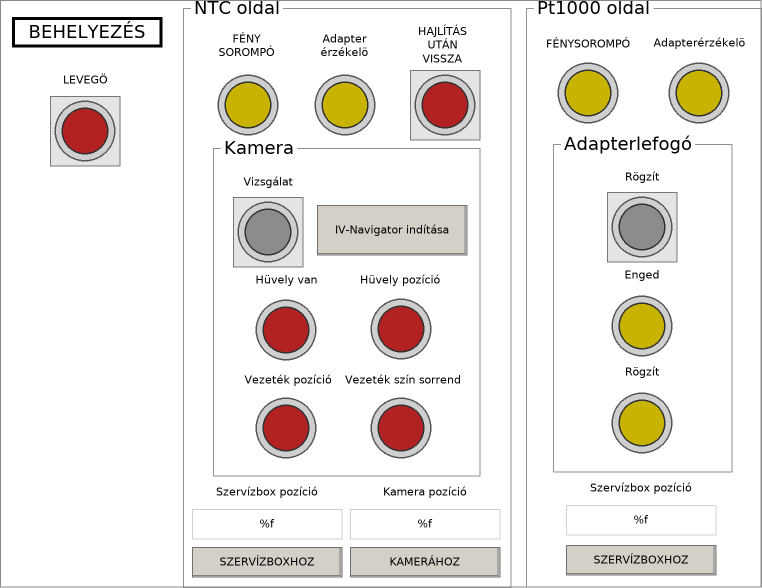
VISUALIZATION Behelyezes  // 762x588
    GroupBox (526,0 236x587), "Pt1000 oldal"
        GroupBox (27,136 179x336), "Adapterlefogó"
            PushSwitch (54,56 70x70), variable: GVL.bAdapterLefogo, behaviour: TOGGLE, style: Switch-PushSwitch-Gray
            Lamp1 (54,155 70x70), variable: GVL.bAdapterLefogoBent, style: Lamp-Lamp1-Yellow
            Lamp1 (54,252 70x70), variable: GVL.bAdapterLefogoKint, style: Lamp-Lamp1-Yellow
            Label (61,226 57x20), "Rögzít"
            Label (62,129 54x20), "Enged"
            Label (60,31 59x20), "Rögzít"
        Lamp1 (138,58 70x70), variable: GVL.bAdaptererzekelo, style: Lamp-Lamp1-Yellow
        Label (122,33 103x20), "Adapterérzékelö"
        Lamp1 (27,58 70x70), variable: GVL.bFenysorompoPt, style: Lamp-Lamp1-Yellow
        Label (10,34 104x20), "FÉNYSOROMPÓ"
        Group (40,478 150x97)
            Button (0,67 150x30), "SZERVÍZBOXHOZ"
                OnMouseUp: execute { PISTITENGELY.lrPistiPosition:=GVL.lrPtSzervizbox; PISTITENGELY.sPistiAxisCommand:='MOVE'; }
            Textfield (0,27 150x30), "%f", text variable: GVL.lrPtSzervizbox
                OnMouseClick: write the text variable via VisuDialogs.Numpad, min -10000, max -1
            Label (0,0 150x20), "Szervízbox pozíció"
    RoundedRectangle (12,17 150x30)
    Label (12,17 150x30), "BEHELYEZÉS"
    GroupBox (183,0 328x588), "NTC oldal"
        GroupBox (30,140 267x336), "Kamera"
            Group (20,32 70x95)
                PushSwitch (0,25 70x70), variable: GVL.bKameraTrigger, behaviour: TOGGLE, style: Switch-PushSwitch-Gray
                Label (2,0 67x20), "Vizsgálat"
            Lamp1 (153,154 70x70), variable: GVL.bKameraHulsePozOK, style: Lamp-Lamp1-Green
            Lamp1 (153,253 70x70), variable: GVL.bKameraSzinekOK, style: Lamp-Lamp1-Green
            Label (130,230 120x20), "Vezeték szín sorrend"
            Label (140,130 94x20), "Hüvely pozíció"
            Lamp1 (153,154 70x70), variable: NOT GVL.bKameraHulsePozOK, invisible if: NOT KAMERA.bVizsgalatKesz OR GVL.bKameraHulsePozOK, style: Lamp-Lamp1-Red
            Lamp1 (153,253 70x70), variable: NOT GVL.bKameraSzinekOK, invisible if: NOT KAMERA.bVizsgalatKesz OR GVL.bKameraSzinekOK, style: Lamp-Lamp1-Red
            Label (30,230 90x20), "Vezeték pozíció"
            Lamp1 (38,253 70x70), variable: GVL.bKameraVezetekPozOK, style: Lamp-Lamp1-Green
            Lamp1 (38,253 70x70), variable: NOT GVL.bKameraVezetekPozOK, invisible if: NOT KAMERA.bVizsgalatKesz OR GVL.bKameraVezetekPozOK, style: Lamp-Lamp1-Red
            Button (104,65 150x50), "IV-Navigator indítása", tooltip "A jelölö lézer saját vezérlö szoftvere", pressed state: Laser.bStartFOBADraw
                OnMouseUp: execute { KAMERA.bStartIVNav:=TRUE; }
            Label (32,130 83x20), "Hüvely van"
            Lamp1 (38,155 70x70), variable: GVL.bKameraHulseVanOK, style: Lamp-Lamp1-Green
            Lamp1 (38,155 70x70), variable: NOT GVL.bKameraHulseVanOK, invisible if: NOT KAMERA.bVizsgalatKesz OR GVL.bKameraHulseVanOK, style: Lamp-Lamp1-Red
        Group (9,482 150x95)
            Textfield (0,27 150x30), "%f", text variable: GVL.lrNTCSzervizbox
                OnMouseClick: write the text variable via VisuDialogs.Numpad, min -10000, max -1
            Button (0,65 150x30), "SZERVÍZBOXHOZ"
                OnMouseUp: execute { JOZSITENGELY.lrJozsiPosition:=GVL.lrNTCSzervizbox; JOZSITENGELY.sJozsiAxisCommand:='MOVE'; }
            Label (0,0 150x20), "Szervízbox pozíció"
        Lamp1 (30,70 70x70), variable: GVL.bFenysorompoNTC, style: Lamp-Lamp1-Yellow
        Label (10,30 107x31), "FÉNY SOROMPÓ"
        Group (167,482 150x95)
            Textfield (0,27 150x30), "%f", text variable: GVL.lrNTCKameraPosition
                OnMouseClick: write the text variable via VisuDialogs.Numpad, min -10000, max -1
            Button (0,65 150x30), "KAMERÁHOZ"
                OnMouseUp: execute { JOZSITENGELY.lrJozsiPosition:=GVL.lrNTCKameraPosition; JOZSITENGELY.sJozsiAxisCommand:='MOVE'; }
            Label (0,0 150x20), "Kamera pozíció"
        Label (110,30 103x31), "Adapter érzékelö"
        Label (220,20 79x50), "HAJLÍTÁS UTÁN VISSZA"
    Label (51,70 69x20), "LEVEGÖ"
    PushSwitch (50,96 70x70), variable: MAIN.bLevego, behaviour: TOGGLE, style: Switch-PushSwitch-Red
    Lamp1 (310,70 70x70), variable: GVL.bNTCAdapterErzekelo, style: Lamp-Lamp1-Yellow
    PushSwitch (410,70 70x70), variable: AUTOMATA.bHajlitasUtanVissza, behaviour: TOGGLE, style: Switch-PushSwitch-Red
END_VISUALIZATION

(* stored: Version 1.1.0.1, ProductVersion 3.1.4024.11
   Visu Behelyezes: Id {e3baf030-60e8-4581-988d-75b2896a3e91} *)
